{attribute 'qualified_only'}
{attribute 'strict'}
TYPE enumColors :
(
	Red := 0,
	Orange := 1,
	Yellow := 2,
	Green := 3,
	Blue := 4,
	Indigo := 5,
	Violet := 6
);
END_TYPE

(* stored: Version 1.1.0.1, ProductVersion 3.1.4024.9
   DUT enumColors: Id {b5b94824-4a8f-4b2b-9329-97d0a87f0724} *)
